FUNCTION_BLOCK PID
  (* Standard: 61499-2 *)
  (* Version 27-01-2014, Gabriel *)
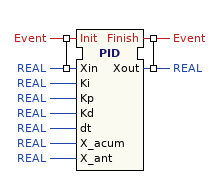
  EVENT_INPUT
    Init WITH Xin;
  END_EVENT
  EVENT_OUTPUT
    Finish WITH Xout;
  END_EVENT
  VAR_INPUT
    Xin : REAL;
    Ki : REAL;
    Kp : REAL;
    Kd : REAL;
    dt : REAL;
    X_acum : REAL := 0;
    X_ant : REAL := 0;
  END_VAR
  VAR_OUTPUT
    Xout : REAL;
  END_VAR
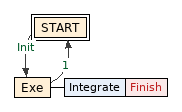
  EC_STATES
    START;
    Exe : Integrate -> Finish;
  END_STATES
  EC_TRANSITIONS
    Exe TO START := 1;
    START TO Exe := Init;
  END_TRANSITIONS
  ALGORITHM Integrate IN Lua:
X_acum = X_acum + Xin*dt         Xout  = Ki*X_acum  + Kp*Xin
  END_ALGORITHM
END_FUNCTION_BLOCK
